// TIA Portal V20 export
DATA_BLOCK "LBP_InternalDB25003"   // DB25003
TITLE = Internal DB for basic program / DB interne pour programme de base
{ S7_Optimized_Access := 'FALSE' }
AUTHOR : SINUMERIK
FAMILY : SINUMERIK_ONE
VERSION : 6.24
// DB only for internal use in the basic program / DB réservé à l'utilisation interne dans le programme de base
// stored: AutoNumber false
   VAR
      traceVar : Struct   // internal use only / réservé à l'utilisation interne
         cmdToPlc { ExternalVisible := 'False'} : Bool;
         identifier { ExternalVisible := 'False'} : UInt;
         symbol { ExternalVisible := 'False'} : WString;
         result { ExternalVisible := 'False'; ExternalWritable := 'False'} : UInt;
         unit { ExternalVisible := 'False'; ExternalWritable := 'False'} : UInt;
         column { ExternalVisible := 'False'; ExternalWritable := 'False'} : UInt;
         row { ExternalVisible := 'False'; ExternalWritable := 'False'} : UInt;
         "type" { ExternalVisible := 'False'; ExternalWritable := 'False'} : UInt;
      END_STRUCT;
   END_VAR
BEGIN
END_DATA_BLOCK
